(* Schneider Machine Expert - Basic project New Grease Machine Twin, file version 2.6.0.0 *)
(* ProjectInformations: Name=New project *)

HARDWARE
  Cpu 0: TM221CE40R
  EthernetConfiguration: NetworkName=M221, IpAllocationMode=FixedAddress, IpAddress=192.168.0.3, SubnetMask=255.255.255.0
  SerialLineConfiguration: Baud=Baud19200, Parity=ParityEven, DataBits=DataBits8, StopBits=StopBits1, PhysicalMedium=PhysicalMediumRs232, TransmissionMode=TransmissionModeModbusRtu, SlaveId=1, Addressing=SlaveAddressing
  MastTask: UsePeriodScanMode=false, PeriodScan=100
  FastTask: Period=255
  CpuBehavior: StartingMode=StartAsPreviousState, AutoSaveRamOnEeprom=true, WatchdogPeriod=250

SYMBOLS  (address, symbol, comment, settings)
  %M0         "RST HMI"
  %M1         "M_BTN START"
  %M2         "M_SENSOR CERTAIN"
  %M3         "M_SENSOR TABLE"
  %M4         "M_BTN CYCLE START"
  %M5         "M_EMG"
  %M6         "M_PROCESS DONE"
  %M7         "M_GREASE EMPTY"
  %M8         "M_GREASE TRIGGER"
  %M9         "M_Q GREASE ACTIVE"
  %M10        "M_Q CERTAIN SENSOR"
  %M11        "M_Q CYCLE START"
  %M12        "M_Q EMERGENCY"
  %M13        "M_Q RED LAMP"
  %M14        "M_Q YELLOW LAMP"
  %M15        "M_Q GREEN LAMP"
  %M16        "M_Q BUZZER"
  %M17        "RED LAMP 2"
  %M18        "TRIGGER YELLOW LAMP"
  %M19        "PAUSE"
  %M20        "FINISH RUN"
  %M21        "RESET BUZZER"
  %M22        "MEMORY M2"
  %M23        "M_POWER MOTOR"
  %M24        "START LAMP BUTTON"
  %M25        "CONTINUE LAMP BUTTON"
  %M26        "M_BASE_ON"
  %M27        "M_TIMER FINISH"
  %M28        "M_STOP_HMI"
  %M29        "REMOVE"
  %M30        "M_START"
  %M31        "M_START_HMI"
  %M32        "SEL_TABLE_ON"
  %M33        "TRIGGER_TABLE"
  %M34        "SEL_TABLE_OFF"
  %M35        "RELEASE HOLD"
  %M36        "ROBOT HOLD"
  %M37        "MAN_GREASE"
  %M38        "TRIGGRER_GREASE"
  %M39        "M_TABLE_SENSOR"
  %M40        "CHECK_GREASE"
  %M41        "RSLT_G_EMPTY"
  %M42        "RSLT_G_NOTEMPTY"
  %M43        "ALARM_ON"
  %M44        "ALARM_OFF"
  %M45        "M_RUN_EMG"
  %M46        "M_TRIG_HOME"
  %M47        "ROBOT_HOME"
  %M48        "M_RESET_MICRO"
  %M49        "POLARITY CHECKED"
  %M50        "NEGATIVE"
  %M51        "POSITIVE"
  %M52        "FIRST RUN"
  %M53        "DONE CUTTING"
  %M54        "NEGATIVE READY"
  %M55        "TRIGGER"
  %M56        "COUNTER OUTPUT"
  %M100       "START GUI"
  %M102       "M_START"
  %MW0        "Count Output"
  %TM0        "TIMER_FINISH"  [Type=TOF, Preset=10, Base=OneSecond]
  %TM1        "ALARM_GREASE"  [Type=TOF, Preset=8, Base=OneSecond]
  %I0.0       "TRIGGER_CLEAN"
  %I0.1       "BTN START"
  %I0.2       "SENSOR CERTAIN"
  %I0.3       "SENSOR TABLE"
  %I0.4       "BTN CYCLE START"
  %I0.5       "BTN EMG"
  %I0.6       "PROCESS DONE"
  %I0.7       "TANK EMPTY"
  %I0.8       "TRIGGER GREASE"
  %I0.9       "MOTOR BASE ON"
  %Q0.0       "GREASE ACTIVE"
  %Q0.1       "CERTAIN SENSOR"
  %Q0.2       "CYCLE START"
  %Q0.3       "EMERGENCY"
  %Q0.4       "RED_LAMP"
  %Q0.5       "YELLOW_LAMP"
  %Q0.6       "GREEN_LAMP"
  %Q0.7       "BUZZER"
  %Q0.8       "POWER_MOTOR"
  %Q0.9       "PB_START_LAMP"
  %Q0.10      "PB_CONTINUE_LAMP"
  %Q0.11      "MOTOR BASE ON(MICRO)"
  %Q0.12      "SELENOID_ON"
  %Q0.13      "CLEAN_NOZZLE"

POU New POU
  (* SectionNumber=1 *)

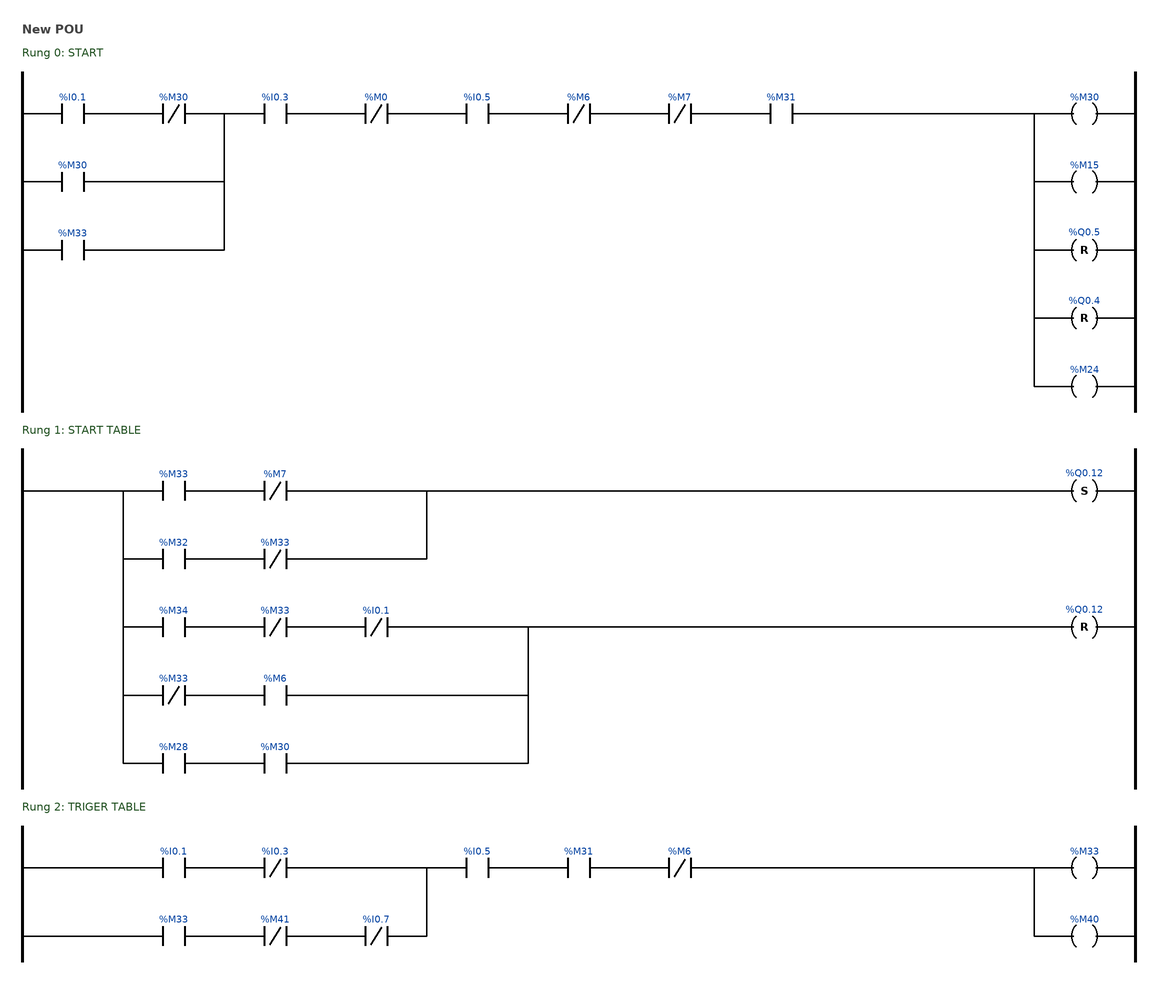

// Rung 0: START
  LD %I0.1
  ANDN %M30
  OR %M30
  OR %M33
  AND %I0.3
  ANDN %M0
  AND %I0.5
  ANDN %M6
  ANDN %M7
  AND %M31
  ST %M30
  ST %M15
  R %Q0.5
  R %Q0.4
  ST %M24
  // as ST:
  //   _t1 := (%I0.1 AND NOT %M30 OR %M30 OR %M33) AND %I0.3 AND NOT %M0 AND %I0.5 AND NOT %M6 AND NOT %M7 AND %M31;
  //   %M30 := _t1;
  //   %M15 := _t1;
  //   IF _t1 THEN %Q0.5 := FALSE; END_IF;
  //   IF _t1 THEN %Q0.4 := FALSE; END_IF;
  //   %M24 := _t1;

// Rung 1: START TABLE
  LD 1
  MPS
  AND( %M33
  ANDN %M7
  OR( %M32
  ANDN %M33
  )
  )
  S %Q0.12
  MPP
  AND( %M34
  ANDN %M33
  ANDN %I0.1
  OR(N %M33
  AND %M6
  )
  OR( %M28
  AND %M30
  )
  )
  R %Q0.12
  // as ST:
  //   IF %M33 AND NOT %M7 OR %M32 AND NOT %M33 THEN %Q0.12 := TRUE; END_IF;
  //   IF %M34 AND NOT %M33 AND NOT %I0.1 OR NOT %M33 AND %M6 OR %M28 AND %M30 THEN %Q0.12 := FALSE; END_IF;

// Rung 2: TRIGER TABLE
  LD %I0.1
  ANDN %I0.3
  OR( %M33
  ANDN %M41
  ANDN %I0.7
  )
  AND %I0.5
  AND %M31
  ANDN %M6
  ST %M33
  ST %M40
  // as ST:
  //   _t1 := (%I0.1 AND NOT %I0.3 OR %M33 AND NOT %M41 AND NOT %I0.7) AND %I0.5 AND %M31 AND NOT %M6;
  //   %M33 := _t1;
  //   %M40 := _t1;

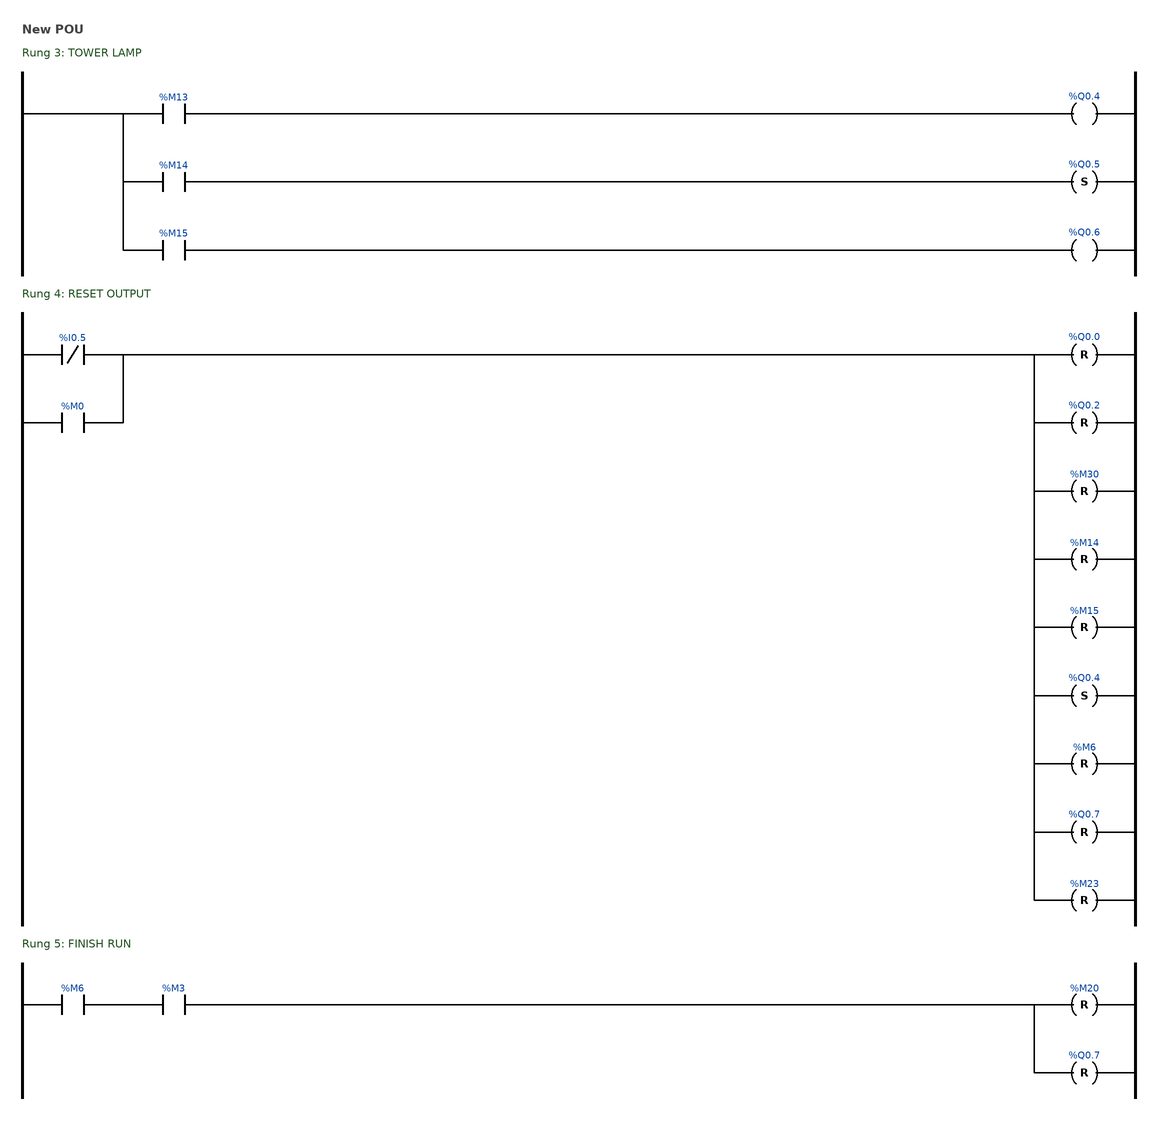

// Rung 3: TOWER LAMP
  LD 1
  MPS
  AND %M13
  ST %Q0.4
  MRD
  AND %M14
  S %Q0.5
  MPP
  AND %M15
  ST %Q0.6
  // as ST:
  //   %Q0.4 := %M13;
  //   IF %M14 THEN %Q0.5 := TRUE; END_IF;
  //   %Q0.6 := %M15;

// Rung 4: RESET OUTPUT
  LDN %I0.5
  OR %M0
  R %Q0.0
  R %Q0.2
  R %M30
  R %M14
  R %M15
  S %Q0.4
  R %M6
  R %Q0.7
  R %M23
  // as ST:
  //   IF NOT %I0.5 OR %M0 THEN %Q0.0 := FALSE; END_IF;
  //   IF NOT %I0.5 OR %M0 THEN %Q0.2 := FALSE; END_IF;
  //   IF NOT %I0.5 OR %M0 THEN %M30 := FALSE; END_IF;
  //   IF NOT %I0.5 OR %M0 THEN %M14 := FALSE; END_IF;
  //   IF NOT %I0.5 OR %M0 THEN %M15 := FALSE; END_IF;
  //   IF NOT %I0.5 OR %M0 THEN %Q0.4 := TRUE; END_IF;
  //   IF NOT %I0.5 OR %M0 THEN %M6 := FALSE; END_IF;
  //   IF NOT %I0.5 OR %M0 THEN %Q0.7 := FALSE; END_IF;
  //   IF NOT %I0.5 OR %M0 THEN %M23 := FALSE; END_IF;

// Rung 5: FINISH RUN
  LD %M6
  AND %M3
  R %M20
  R %Q0.7
  // as ST:
  //   IF %M6 AND %M3 THEN %M20 := FALSE; END_IF;
  //   IF %M6 AND %M3 THEN %Q0.7 := FALSE; END_IF;

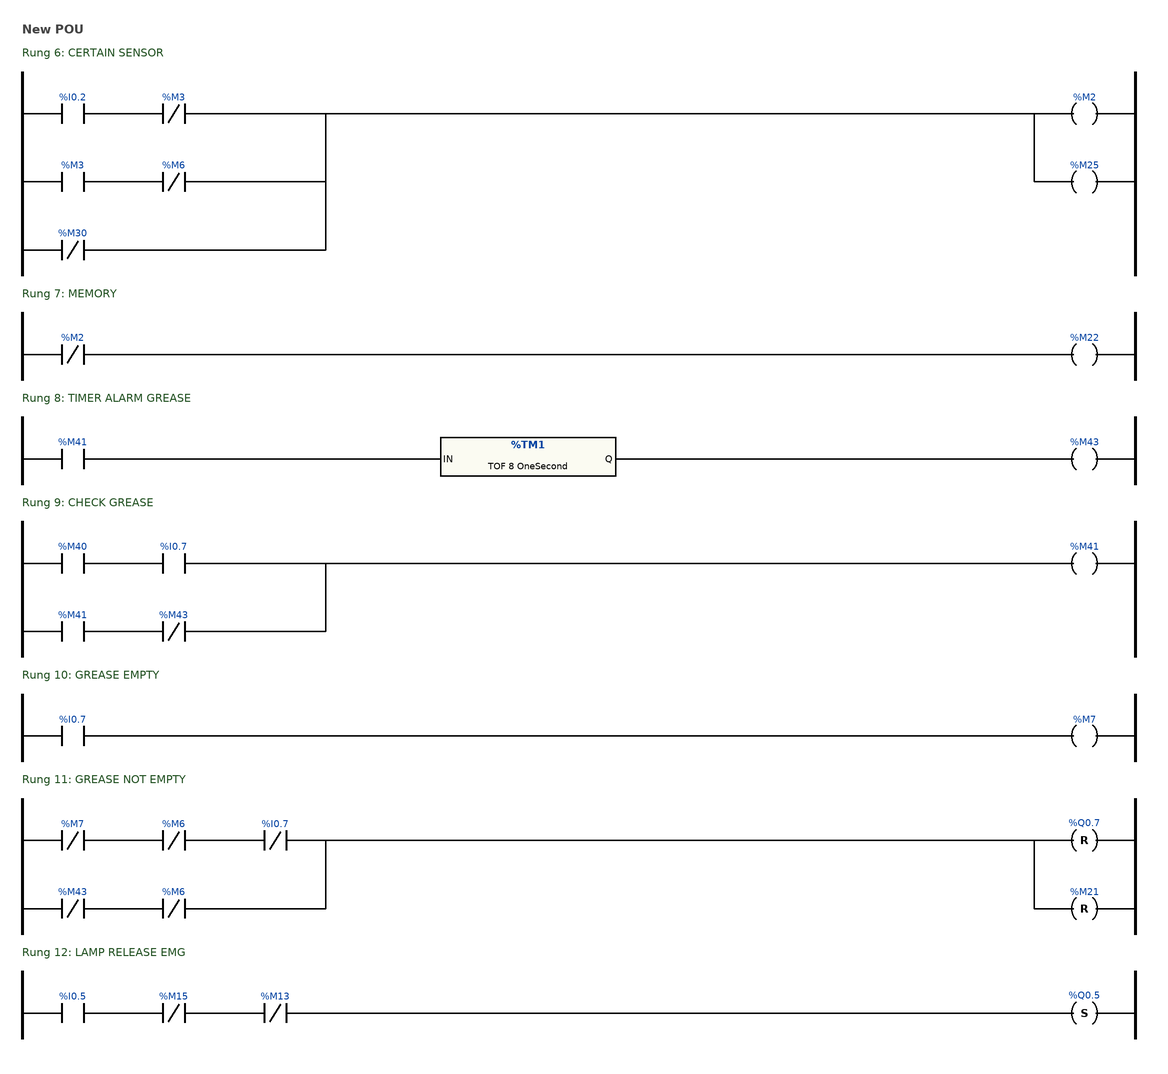

// Rung 6: CERTAIN SENSOR
  LD %I0.2
  ANDN %M3
  OR( %M3
  ANDN %M6
  )
  ORN %M30
  ST %M2
  ST %M25
  // as ST:
  //   %M2 := %I0.2 AND NOT %M3 OR %M3 AND NOT %M6 OR NOT %M30;
  //   %M25 := %I0.2 AND NOT %M3 OR %M3 AND NOT %M6 OR NOT %M30;

// Rung 7: MEMORY
  LDN %M2
  ST %M22
  // as ST:
  //   %M22 := NOT %M2;

// Rung 8: TIMER ALARM GREASE
  BLK %TM1
  LD %M41
  IN
  OUT_BLK
  LD Q
  ST %M43
  END_BLK
  // as ST:
  //   %TM1(IN := %M41);
  //   %M43 := %TM1.Q;

// Rung 9: CHECK GREASE
  LD %M40
  AND %I0.7
  OR( %M41
  ANDN %M43
  )
  ST %M41
  // as ST:
  //   %M41 := %M40 AND %I0.7 OR %M41 AND NOT %M43;

// Rung 10: GREASE EMPTY
  LD %I0.7
  ST %M7
  // as ST:
  //   %M7 := %I0.7;

// Rung 11: GREASE NOT EMPTY
  LDN %M7
  ANDN %M6
  ANDN %I0.7
  OR(N %M43
  ANDN %M6
  )
  R %Q0.7
  R %M21
  // as ST:
  //   IF NOT %M7 AND NOT %M6 AND NOT %I0.7 OR NOT %M43 AND NOT %M6 THEN %Q0.7 := FALSE; END_IF;
  //   IF NOT %M7 AND NOT %M6 AND NOT %I0.7 OR NOT %M43 AND NOT %M6 THEN %M21 := FALSE; END_IF;

// Rung 12: LAMP RELEASE EMG
  LD %I0.5
  ANDN %M15
  ANDN %M13
  S %Q0.5
  // as ST:
  //   IF %I0.5 AND NOT %M15 AND NOT %M13 THEN %Q0.5 := TRUE; END_IF;

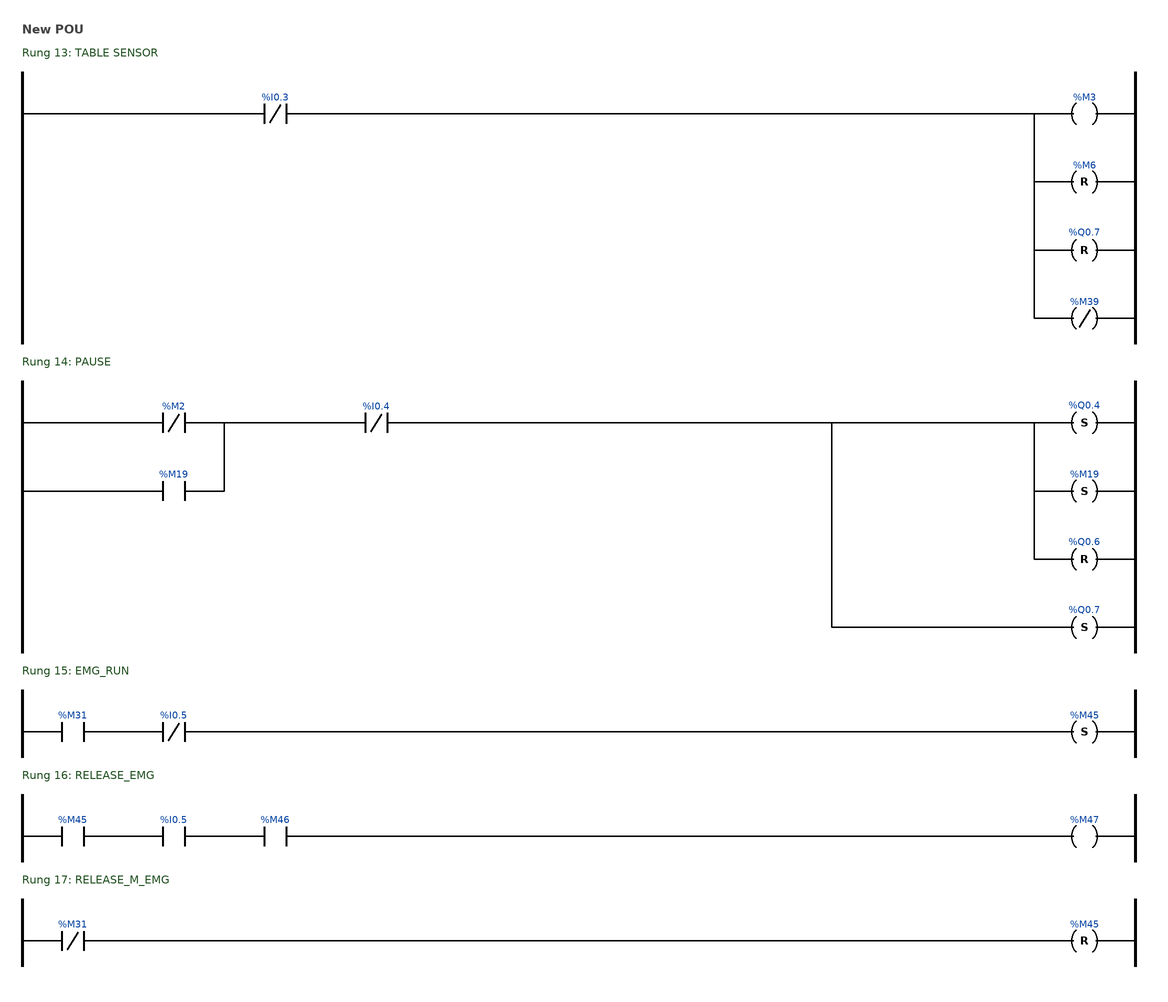

// Rung 13: TABLE SENSOR
  LDN %I0.3
  ST %M3
  R %M6
  R %Q0.7
  STN %M39
  // as ST:
  //   %M3 := NOT %I0.3;
  //   IF NOT %I0.3 THEN %M6 := FALSE; END_IF;
  //   IF NOT %I0.3 THEN %Q0.7 := FALSE; END_IF;
  //   %M39 := NOT (NOT %I0.3);

// Rung 14: PAUSE
  LDN %M2
  OR %M19
  ANDN %I0.4
  S %Q0.4
  S %M19
  R %Q0.6
  S %Q0.7
  // as ST:
  //   IF (NOT %M2 OR %M19) AND NOT %I0.4 THEN %Q0.4 := TRUE; END_IF;
  //   _t1 := (NOT %M2 OR %M19) AND NOT %I0.4;
  //   IF _t1 THEN %M19 := TRUE; END_IF;
  //   IF _t1 THEN %Q0.6 := FALSE; END_IF;
  //   IF _t1 THEN %Q0.7 := TRUE; END_IF;

// Rung 15: EMG_RUN
  LD %M31
  ANDN %I0.5
  S %M45
  // as ST:
  //   IF %M31 AND NOT %I0.5 THEN %M45 := TRUE; END_IF;

// Rung 16: RELEASE_EMG
  LD %M45
  AND %I0.5
  AND %M46
  ST %M47
  // as ST:
  //   %M47 := %M45 AND %I0.5 AND %M46;

// Rung 17: RELEASE_M_EMG
  LDN %M31
  R %M45
  // as ST:
  //   IF NOT %M31 THEN %M45 := FALSE; END_IF;

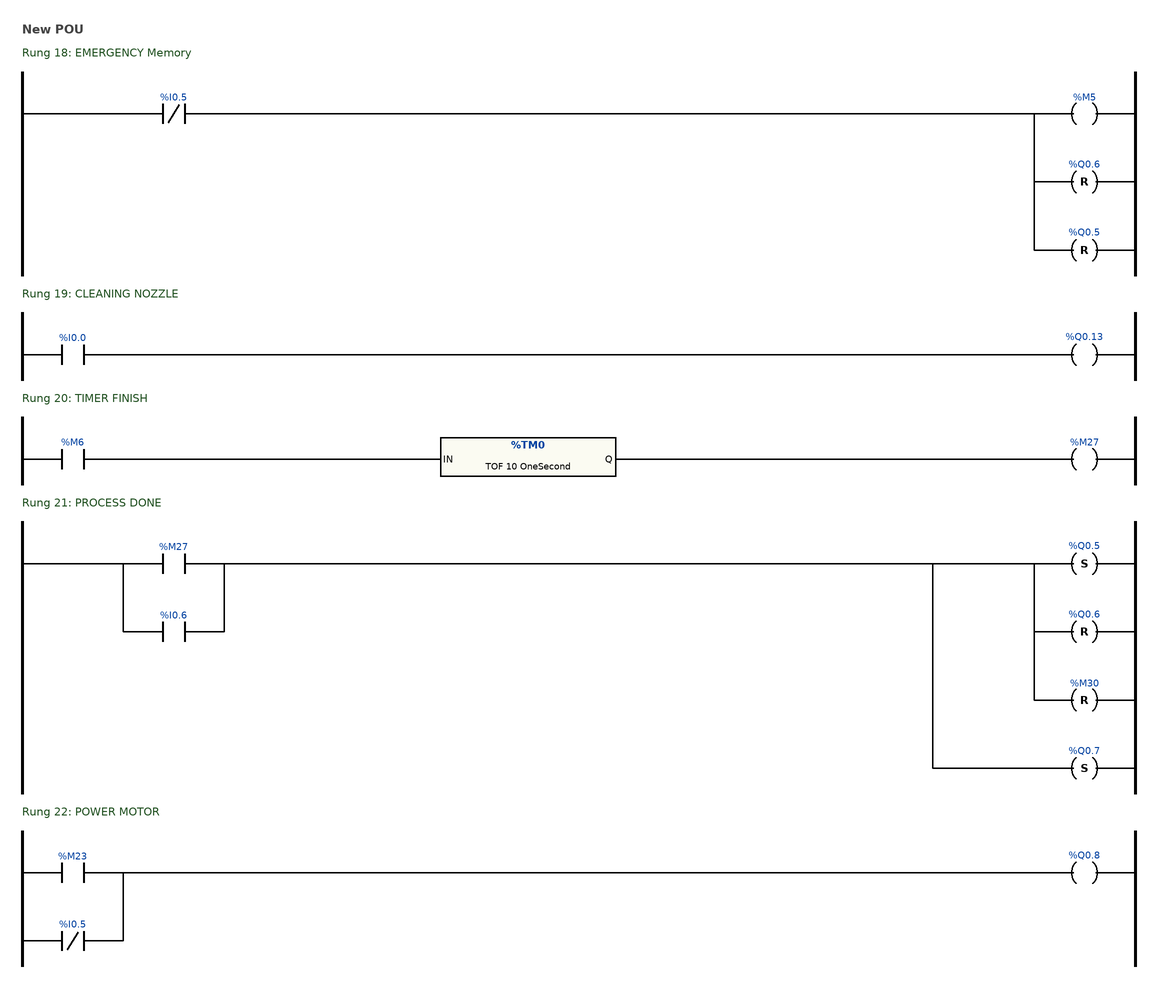

// Rung 18: EMERGENCY Memory
  LDN %I0.5
  ST %M5
  R %Q0.6
  R %Q0.5
  // as ST:
  //   %M5 := NOT %I0.5;
  //   IF NOT %I0.5 THEN %Q0.6 := FALSE; END_IF;
  //   IF NOT %I0.5 THEN %Q0.5 := FALSE; END_IF;

// Rung 19: CLEANING NOZZLE
  LD %I0.0
  ST %Q0.13
  // as ST:
  //   %Q0.13 := %I0.0;

// Rung 20: TIMER FINISH
  BLK %TM0
  LD %M6
  IN
  OUT_BLK
  LD Q
  ST %M27
  END_BLK
  // as ST:
  //   %TM0(IN := %M6);
  //   %M27 := %TM0.Q;

// Rung 21: PROCESS DONE
  LD 1
  AND( %M27
  OR %I0.6
  )
  S %Q0.5
  R %Q0.6
  R %M30
  S %Q0.7
  // as ST:
  //   IF %M27 OR %I0.6 THEN %Q0.5 := TRUE; END_IF;
  //   IF %M27 OR %I0.6 THEN %Q0.6 := FALSE; END_IF;
  //   IF %M27 OR %I0.6 THEN %M30 := FALSE; END_IF;
  //   IF %M27 OR %I0.6 THEN %Q0.7 := TRUE; END_IF;

// Rung 22: POWER MOTOR
  LD %M23
  ORN %I0.5
  ST %Q0.8
  // as ST:
  //   %Q0.8 := %M23 OR NOT %I0.5;

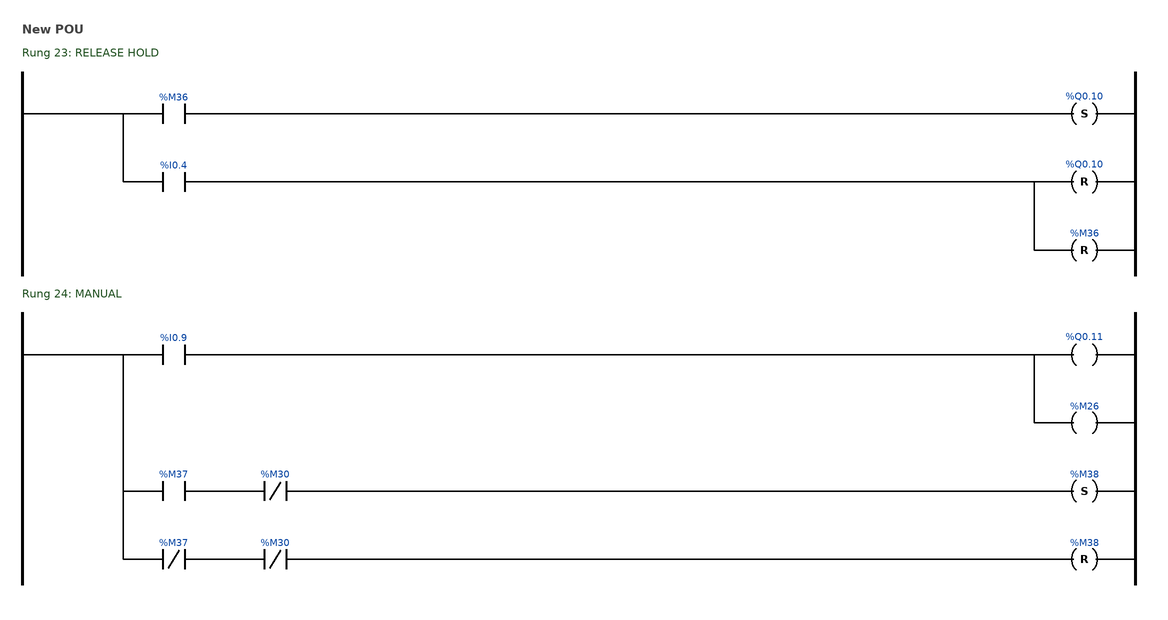

// Rung 23: RELEASE HOLD
  LD 1
  MPS
  AND %M36
  S %Q0.10
  MPP
  AND %I0.4
  R %Q0.10
  R %M36
  // as ST:
  //   IF %M36 THEN %Q0.10 := TRUE; END_IF;
  //   IF %I0.4 THEN %Q0.10 := FALSE; END_IF;
  //   IF %I0.4 THEN %M36 := FALSE; END_IF;

// Rung 24: MANUAL
  LD 1
  MPS
  AND %I0.9
  ST %Q0.11
  ST %M26
  MRD
  AND %M37
  ANDN %M30
  S %M38
  MPP
  ANDN %M37
  ANDN %M30
  R %M38
  // as ST:
  //   %Q0.11 := %I0.9;
  //   %M26 := %I0.9;
  //   IF %M37 AND NOT %M30 THEN %M38 := TRUE; END_IF;
  //   IF NOT %M37 AND NOT %M30 THEN %M38 := FALSE; END_IF;

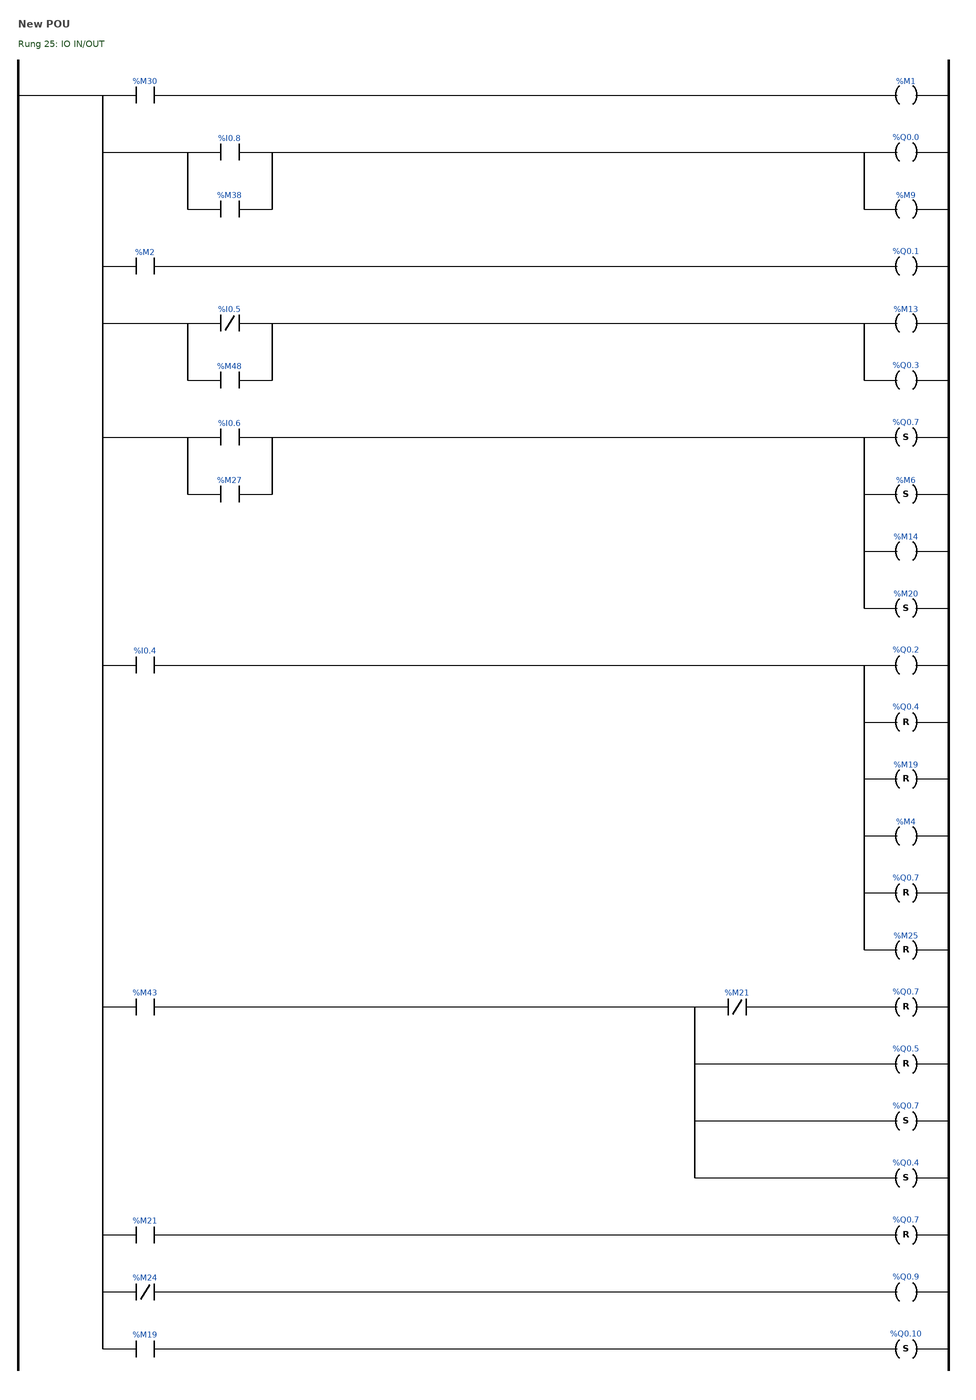

// Rung 25: IO IN/OUT
  LD 1
  MPS
  AND %M30
  ST %M1
  MRD
  AND( %I0.8
  OR %M38
  )
  ST %Q0.0
  ST %M9
  MRD
  AND %M2
  ST %Q0.1
  MRD
  AND(N %I0.5
  OR %M48
  )
  ST %M13
  ST %Q0.3
  MRD
  AND( %I0.6
  OR %M27
  )
  S %Q0.7
  S %M6
  ST %M14
  S %M20
  MRD
  AND %I0.4
  ST %Q0.2
  R %Q0.4
  R %M19
  ST %M4
  R %Q0.7
  R %M25
  MRD
  AND %M43
  MPS
  ANDN %M21
  R %Q0.7
  MRD
  R %Q0.5
  MRD
  S %Q0.7
  MPP
  S %Q0.4
  MRD
  AND %M21
  R %Q0.7
  MRD
  ANDN %M24
  ST %Q0.9
  MPP
  AND %M19
  S %Q0.10
  // as ST:
  //   %M1 := %M30;
  //   %Q0.0 := %I0.8 OR %M38;
  //   %M9 := %I0.8 OR %M38;
  //   %Q0.1 := %M2;
  //   %M13 := NOT %I0.5 OR %M48;
  //   %Q0.3 := NOT %I0.5 OR %M48;
  //   IF %I0.6 OR %M27 THEN %Q0.7 := TRUE; END_IF;
  //   IF %I0.6 OR %M27 THEN %M6 := TRUE; END_IF;
  //   %M14 := %I0.6 OR %M27;
  //   IF %I0.6 OR %M27 THEN %M20 := TRUE; END_IF;
  //   %Q0.2 := %I0.4;
  //   IF %I0.4 THEN %Q0.4 := FALSE; END_IF;
  //   IF %I0.4 THEN %M19 := FALSE; END_IF;
  //   %M4 := %I0.4;
  //   IF %I0.4 THEN %Q0.7 := FALSE; END_IF;
  //   IF %I0.4 THEN %M25 := FALSE; END_IF;
  //   IF %M43 AND NOT %M21 THEN %Q0.7 := FALSE; END_IF;
  //   IF %M43 THEN %Q0.5 := FALSE; END_IF;
  //   IF %M43 THEN %Q0.7 := TRUE; END_IF;
  //   IF %M43 THEN %Q0.4 := TRUE; END_IF;
  //   IF %M21 THEN %Q0.7 := FALSE; END_IF;
  //   %Q0.9 := NOT %M24;
  //   IF %M19 THEN %Q0.10 := TRUE; END_IF;
